FUNCTION_BLOCK FB_Start
VAR_INPUT
	bSwitchOn				: BOOL;
	bSwitchOff				: BOOL;
END_VAR
VAR
	bSwitchedOn				: BOOL;
END_VAR

{attribute 'TcRpcEnable'}
METHOD SwitchOff
bSwitchedOn := FALSE;
END_METHOD

{attribute 'TcRpcEnable'}
METHOD SwitchOn : BOOL
VAR_INPUT
END_VAR
bSwitchedOn := TRUE;
END_METHOD

END_FUNCTION_BLOCK

(* stored: Version 1.1.0.1, ProductVersion 3.1.4024.11
   POU FB_Start: Id {691bad33-fd39-49a6-b5a9-a63fb496f0d3}, SpecialFunc None
   Method SwitchOff: Id {66067207-5224-40d9-9f3e-1736f1f2e435}
   Method SwitchOn: Id {9cf239e1-6394-4059-b552-285229f77b77} *)
